//==================================================================================================
//								RJM Maszyny sp. z o.o.
//									04.02.2022
//	Obsługa elektrozaworu 3/2 normalnie zamkniętego
// 	v1.0	|| TC v 3.1.4024.22		|| - pierwsza wersja
//==================================================================================================
FUNCTION_BLOCK FB_Elektrozawor_3na2_NC IMPLEMENTS I_Elektrozawor_3na2
VAR
	fbCewka									: FB_ElektrozaworCewka;
END_VAR

//==================================================================================================
//								RJM Maszyny sp. z o.o.
//									04.02.2022
//	Włączenie cewki - wyjscie 2
// 	v1.0	|| TC v 3.1.4024.22		|| - pierwsza wersja
//==================================================================================================
METHOD Wlacz
VAR_INPUT
END_VAR
fbCewka.Wylacz ();
END_METHOD

//==================================================================================================
//								RJM Maszyny sp. z o.o.
//									04.02.2022
//	Wyłączenie cewki - wyjscie 2
// 	v1.0	|| TC v 3.1.4024.22		|| - pierwsza wersja
//==================================================================================================
METHOD Wylacz
VAR_INPUT
END_VAR
fbCewka.Wlacz ();
END_METHOD

END_FUNCTION_BLOCK

(* stored: Version 1.1.0.1, ProductVersion 3.1.4024.11
   POU FB_Elektrozawor_3na2_NC: Id {da48c5f4-04a0-486f-a944-3e5ba1447a55}, SpecialFunc None
   Method Wlacz: Id {0a38aa95-1740-41f9-a5b8-c999ceaa5f76}
   Method Wylacz: Id {148ac881-0ef0-40d2-8eb5-022c7e308737} *)
